# B&R Automation Studio project FeederLib (part 2)

#### FBFeeder.st
```iecst
(* TODO: Add your comment here *)
FUNCTION_BLOCK FBFeeder
	IF Enable THEN
		CASE Status OF
			FEED_ERROR:
			FEED_INIT:
				FBControl.Enable := TRUE;
				FBControl.TareK := Config.DefaultTareK;

				TON_BufferDelay.PT := Config.BufferDelay;
				TON_TareCalcDelay.PT := Config.TareCalcDelay;
				TON_DeviationCalcDelay.PT := Config.DeviationCalcDelay;
				TON_ToGoToAutoDelay.PT := Config.ToGoToAutoDelay;

				i := 0;
				j := 0;

				UserInfo.Rate := 0;
				UserInfo.TareK := 0;
				UserInfo.Deviation := 0;
				IF FBControl.Status = FEEDCTRL_READY_TO_FEED THEN
					Status := FEED_READY;
				END_IF
			FEED_READY:
				IF Start THEN
					FBControl.Start := TRUE;
				END_IF
				IF Reset THEN
					Status := FEED_RESET;
				END_IF
				IF FBControl.Status = FEEDCTRL_FEEDING THEN
					Status := FEED_FEEDING;
				END_IF
			FEED_FEEDING:
				IF Start THEN
					TON_WriteInBufferPeriod.IN := TRUE;
					TON_WriteInBufferPeriod();
					IF TON_WriteInBufferPeriod.Q THEN
						TON_WriteInBufferPeriod.IN := FALSE;
						IF NOT WriteInWTP THEN
							// задержка заполнения буфферов W T P
							TON_BufferDelay.IN := TRUE;
							TON_BufferDelay();
							IF TON_BufferDelay.Q THEN
								WriteInWTP := TRUE;
								TON_BufferDelay.IN := FALSE;
							END_IF
						ELSE
							// заполнение буфера W T P
							WBuffer[i] := UserInfo.Weight;
							IF i = 0 THEN
								PBuffer[0] := PBuffer[2399] + FBControl.UserInfo.ActualSpeed/100000;
								TBuffer[0] := TBuffer[2399] + 0.1;
							ELSE
								PBuffer[i] := PBuffer[i-1] + FBControl.UserInfo.ActualSpeed/100000;
								TBuffer[i] := TBuffer[i-1] + 0.1;
							END_IF

							IF i = 2399 THEN
								i := 0;
								RewriteWTP := TRUE;
							ELSE
								i := i + 1;
							END_IF

							IF NOT WriteInTareK THEN
								// задержка заполнения буффера тарировочного коэффициента
								TON_TareCalcDelay.IN := TRUE;
								TON_TareCalcDelay();
								IF TON_TareCalcDelay.Q THEN
									WriteInTareK := TRUE;
									TON_TareCalcDelay.IN := FALSE;
								END_IF
							ELSE
								// заполнение буффера тарировочного коэффициента
								IF RewriteWTP THEN
									UserInfo.TareK := USINT_TO_REAL(Config.Handler.Ratio)*FFeederRatio(ADR(WBuffer),ADR(PBuffer),ADR(TBuffer),2399)/0.6;
								ELSE
									UserInfo.TareK := USINT_TO_REAL(Config.Handler.Ratio)*FFeederRatio(ADR(WBuffer),ADR(PBuffer),ADR(TBuffer),i)/0.6;
								END_IF
								TareKBuffer[j] := UserInfo.TareK;

								IF j = 2399 THEN
									j := 0;
									RewriteTareK := TRUE;
								ELSE
									j := j + 1;
								END_IF

								IF NOT CalcDeviation THEN
									// задержка расчета стандартной погрешности татировочного коэффициента
									TON_DeviationCalcDelay.IN := TRUE;
									TON_DeviationCalcDelay();
									IF TON_DeviationCalcDelay.Q THEN
										CalcDeviation := TRUE;
										TON_DeviationCalcDelay.IN := FALSE;
									END_IF
								ELSE
									// расчет стандартного откланения погрешности тарировочного коэффициента
									IF RewriteTareK THEN
										UserInfo.Deviation := FStdDeviation(ADR(TareKBuffer),2399);
									ELSE
										UserInfo.Deviation := FStdDeviation(ADR(TareKBuffer),j);
									END_IF
								END_IF
							END_IF
						END_IF
					END_IF
					// Выбор тарировочного коэффициента в зависимости от конфигурации
					IF Control.ManualTareControl THEN
						FBControl.TareK := Control.TareK;
					ELSE
						IF NOT UserInfo.IsAUTO THEN
							FBControl.TareK := Config.DefaultTareK;
							IF CalcDeviation THEN
								IF (UserInfo.Deviation <> 0) AND (UserInfo.Deviation < Config.DeviationLimit) THEN
									TON_ToGoToAutoDelay.IN := TRUE;
									IF TON_ToGoToAutoDelay.Q THEN
										UserInfo.IsAUTO := TRUE;
										TON_ToGoToAutoDelay.IN := FALSE;
									END_IF;
								ELSE
									TON_ToGoToAutoDelay.IN := FALSE;
									FBControl.TareK := Config.DefaultTareK;
								END_IF
								TON_ToGoToAutoDelay();
							ELSE
								FBControl.TareK := Config.DefaultTareK;
							END_IF
						ELSE
							IF UserInfo.Deviation < Config.DeviationLimit THEN
								UserInfo.IsAUTO := FALSE;
							ELSE
								FBControl.TareK := UserInfo.TareK;
							END_IF
						END_IF
					END_IF
				ELSE
					FBControl.Start := FALSE;
					Status := FEED_PAUSE;
				END_IF
			FEED_RESET:
				FOR i := 0 TO 2399 DO
					WBuffer[i] := 0;
					TBuffer[i] := 0;
					PBuffer[i] := 0;
					TareKBuffer[i] := 0;
				END_FOR
				i := 0;
				j := 0;

				RewriteWTP := FALSE;
				RewriteTareK := FALSE;
				WriteInWTP := FALSE;
				WriteInTareK := FALSE;
				CalcDeviation := FALSE;
				UserInfo.IsAUTO := FALSE;

				Reset := FALSE;
				Status := FEED_READY;

				UserInfo.Rate := 0;
				UserInfo.TareK := 0;
				UserInfo.Deviation := 0;
			FEED_PAUSE:
				IF Start THEN
					Status := FEED_READY;
					IF RewriteWTP THEN
						IF i = 0 THEN
							IF ABS(WBuffer[2399]-UserInfo.Weight) > Config.ResetWeightLimit THEN
								Status := FEED_RESET;
							END_IF
						ELSE
							IF ABS(WBuffer[i-1]-UserInfo.Weight) > Config.ResetWeightLimit THEN
								Status := FEED_RESET;
							END_IF
						END_IF
					ELSE
						IF (i <> 0) AND (ABS(WBuffer[i-1]-UserInfo.Weight) > Config.ResetWeightLimit) THEN
							Status := FEED_RESET;
						END_IF
					END_IF
				END_IF
		END_CASE
		FBControl.Config := Config.Handler;
		FBControl.Control := Control.Handler;
		FBControl.IOin := IOin.Handler;
		FBControl();
		UserInfo.Handler := FBControl.UserInfo;
		UserInfo.Weight := CalibrateREAL(DINT_TO_REAL(IOin.aiWeight), Config.WeightCalibrate);
		UserInfo.Rate := FBControl.UserInfo.ActualSpeed*UserInfo.TareK*0.6/USINT_TO_REAL(Config.Handler.Ratio);
		IOout := FBControl.IOout;
	ELSE
		Status := FEED_INIT;
	END_IF
END_FUNCTION_BLOCK
```

#### FBFeederHandler.st
```iecst
(* TODO: Add your comment here *)
FUNCTION_BLOCK FBFeederHandler
	IF Enable THEN
		CASE Status OF
			FEEDCTRL_ERROR:
				// error case
			FEEDCTRL_INIT:
				AxisBasic.MpLink := Config.AxisConfigLink;
				AxisBasic.Enable := TRUE;
				AxisBasic.Parameters := Config.AxisBasicParLink;
				AxisBasic.Axis := Config.ACPConfigLink;

				AxisCyclicSet.MpLink := Config.AxisConfigLink;
				AxisCyclicSet.Enable := TRUE;
				AxisCyclicSet.Parameters := Config.AxisCyclicSetParLink;

				IF (AxisBasic.Active) THEN
					UserInfo.Active := TRUE;
					AxisBasic.Power := 1;
					IF (AxisBasic.PowerOn) THEN
						IF (AxisBasic.IsHomed = 0) THEN
							AxisBasic.Home := 1;
						ELSE
							AxisBasic.Home := 0;
							IF (AxisCyclicSet.Active) THEN
								AxisCyclicSet.CyclicVelocity := 1;
								Status := FEEDCTRL_READY_TO_FEED;
							END_IF
						END_IF
					END_IF
				END_IF

			FEEDCTRL_READY_TO_FEED:
				IF (Start) THEN
					Status := FEEDCTRL_PREPURGE;
				END_IF

				IOout.aoGasRate := 0;
				IOout.doShutOff := TRUE;
				IOout.doMixer := FALSE;
			FEEDCTRL_PREPURGE:
				IF (Start) THEN
					IF (TON_Prepurge.Q) THEN
						TON_Prepurge.IN := 0;
						Status := FEEDCTRL_FEEDING;
					ELSE
						TON_Prepurge.IN := 1;
					END_IF
				ELSE
					TON_Prepurge.IN := 0;
					Status := FEEDCTRL_READY_TO_FEED;
				END_IF
				TON_Prepurge(PT := Config.PrepurgeTime);

				IOout.aoGasRate := Calibrate(Control.GasRate,Config.GasCalibrateOut);
				IOout.doShutOff := FALSE;
				IOout.doMixer := TRUE;
			FEEDCTRL_FEEDING:
				IF (Start) THEN
					AxisCyclicSet.Velocity := ((LIMIT(0,(Control.PowderRate/(TareK*10)),100)*(100+Control.KZU))/Control.KZP)*Config.Ratio/0.6;
				ELSE
					AxisCyclicSet.Velocity := 0;
					Status := FEEDCTRL_POSTPURGE;
				END_IF

				IOout.aoGasRate := Calibrate(Control.GasRate,Config.GasCalibrateOut);
			FEEDCTRL_POSTPURGE:
				IF (Start) THEN
					TON_Postpurge.IN := 0;
					Status := FEEDCTRL_FEEDING;
				ELSE
					IF (TON_Postpurge.Q) THEN
						TON_Postpurge.IN := 0;
						Status := FEEDCTRL_READY_TO_FEED;
					ELSE
						TON_Postpurge.IN := 1;
					END_IF
				END_IF
				TON_Postpurge(PT := Config.PostpurgeTime);

				IOout.aoGasRate := Calibrate(Control.GasRate,Config.GasCalibrateOut);
		END_CASE
		// добавить проверку чтобы AxisConfigLink != 0
		AxisBasic();
		AxisCyclicSet();

		UserInfo.ActualSpeed := AxisBasic.Velocity;
	END_IF

END_FUNCTION_BLOCK
```

#### FBSpendTotalizer.st
```iecst
(* TODO: Add your comment here *)
FUNCTION_BLOCK FBSpendTotalizer

	CASE Status OF
		SPENDTOTALIZER_INIT:
			TON_WeightCheckPeriod.PT := Period;
			Status := SPENDTOTALIZER_WAIT;
		SPENDTOTALIZER_BIZY:
			TON_WeightCheckPeriod();
			IF TON_WeightCheckPeriod.Q THEN
				IF ((TempVal - Weight) > Delta) AND ((TempVal - Weight) > 0) THEN
					CounterLink := CounterLink + (TempVal - Weight);
					TempVal := Weight;
				END_IF
				TON_WeightCheckPeriod.IN := FALSE;
				TON_WeightCheckPeriod();
				TON_WeightCheckPeriod.IN := TRUE;
			END_IF
			IF NOT Active THEN
				IF ((TempVal - Weight) < Delta) AND ((TempVal - Weight) > 0) THEN
					CounterLink := CounterLink + (TempVal - Weight);
					TempVal := Weight;
				END_IF
				TON_WeightCheckPeriod.IN := FALSE;
				TON_WeightCheckPeriod();
				Status := SPENDTOTALIZER_PAUSE;
			END_IF
		SPENDTOTALIZER_PAUSE:
			IF Active THEN
				IF (ABS(TempVal - Weight) > 10*Delta) THEN
					Status := SPENDTOTALIZER_WAIT;
				ELSE
					Status := SPENDTOTALIZER_BIZY;
				END_IF
			END_IF
			TON_WeightCheckPeriod.IN := TRUE;
		SPENDTOTALIZER_WAIT:
			IF Active THEN
				TempVal := Weight;
				Status := SPENDTOTALIZER_BIZY;
			END_IF
	END_CASE

END_FUNCTION_BLOCK
```

#### FBFeederControl.st - not listed in the package file held
```iecst
(* TODO: Add your comment here *)
FUNCTION_BLOCK FBFeederControl
	IF Enable THEN
		CASE Status OF
			FEEDCTRL_ERROR:
				// error case
			FEEDCTRL_INIT:
				// добавить проверку чтобы AxisConfigLink != 0
				AxisBasic.MpLink := Config.AxisConfigLink;
				AxisBasic.Enable := TRUE;
				AxisBasic.Parameters := Config.AxisBasicParLink;
				AxisBasic.Axis := Config.ACPConfigLink;

				AxisCyclicSet.MpLink := Config.AxisConfigLink;
				AxisCyclicSet.Enable := TRUE;
				AxisCyclicSet.Parameters := Config.AxisCyclicSetParLink;

				IF (AxisBasic.Active) THEN
					UserInfo.Active := TRUE;
					AxisBasic.Power := 1;
					IF (AxisBasic.PowerOn) THEN
						IF (AxisBasic.IsHomed = 0) THEN
							AxisBasic.Home := 1;
						ELSE
							AxisBasic.Home := 0;
							IF (AxisCyclicSet.Active) THEN
								AxisCyclicSet.CyclicVelocity := 1;
								Status := FEEDCTRL_READY_TO_FEED;
							END_IF;
						END_IF;
					END_IF;
				END_IF;
			FEEDCTRL_READY_TO_FEED:
				IF (Start) THEN
					Status := FEEDCTRL_PREPURGE;
				END_IF

				IO.Out.aoGasRate := 0;
				IO.Out.doShutOff := TRUE;
				IO.Out.doMixer := FALSE;
			FEEDCTRL_PREPURGE:
				IF (Start) THEN
					IF (TON_Prepurge.Q) THEN
						TON_Prepurge.IN := 0;
						Status := FEEDCTRL_FEEDING;
					ELSE
						TON_Prepurge.IN := 1;
					END_IF
				ELSE
					TON_Prepurge.IN := 0;
					Status := FEEDCTRL_READY_TO_FEED;
				END_IF
				TON_Prepurge(PT := Config.PrepurgeTime);

				IO.Out.aoGasRate := Calibrate(Control.GasRate,Config.GasCalibrateOut);
				IO.Out.doShutOff := FALSE;
				IO.Out.doMixer := TRUE;
			FEEDCTRL_FEEDING:
				IF (Start) THEN
					AxisCyclicSet.Velocity := ((Control.PowderRate*(100+Control.KZU))/Control.KZP)*TareK;
				ELSE
					AxisCyclicSet.Velocity := 0;
					Status := FEEDCTRL_POSTPURGE;
				END_IF

				IO.Out.aoGasRate := Calibrate(Control.GasRate,Config.GasCalibrateOut);
			FEEDCTRL_POSTPURGE:
				IF (Start) THEN
					TON_Postpurge.IN := 0;
					Status := FEEDCTRL_FEEDING;
				ELSE
					IF (TON_Postpurge.Q) THEN
						TON_Postpurge.IN := 0;
						Status := FEEDCTRL_READY_TO_FEED;
					ELSE
						TON_Postpurge.IN := 1;
					END_IF
				END_IF
				TON_Postpurge(PT := Config.PostpurgeTime);

				IO.Out.aoGasRate := Calibrate(Control.GasRate,Config.GasCalibrateOut);
		END_CASE
		AxisBasic();
		AxisCyclicSet();
		UserInfo.ActualSpeed := AxisBasic.Velocity;
	END_IF

END_FUNCTION_BLOCK
```

#### FLinearRegrationKoef.st - not listed in the package file held
```iecst
(* TODO: Add your comment here *)
FUNCTION FLinearRegrationKoef
	sumx := 0;
	sumy := 0;
	sump := 0;
	sumx2 := 0;
	sumxy := 0;
	sumxp := 0;

	FOR i := 0 TO n-1 DO
		weight ACCESS (weightArrayAdr + 32*i);
		position ACCESS (positionArrayAdr + 32*i);
		sumy := sumy + weight;
		sump := sump + position;
		sumxy := sumxy + (i*weight);
		sumxp := sumxp + (i*position);
	END_FOR
	sumx := (lengthOfArray*(lengthOfArray+1))/2;
	sumx2 := (lengthOfArray*(lengthOfArray+1)*(2*lengthOfArray+1))/6;

	sxx := sumx2 - (sumx*sumx)/UINT_TO_REAL(n);
	sxy := sumxy - (sumx*sumy)/UINT_TO_REAL(n);
	sxp := sumxp - (sumx*sump)/UINT_TO_REAL(n);
	k := sxy/sxx;
	kp := sxp/sxx;

	FLinearRegrationKoef := (-k*60)/kp;
END_FUNCTION
```

#### FRatePerMinute.st - not listed in the package file held
```iecst
(* TODO: Add your comment here *)
FUNCTION FRatePerMinute
	sumx := 0;
	sumy := 0;
	sump := 0;
	sumx2 := 0;
	sumxy := 0;
	sumxp := 0;

	FOR i := 0 TO lengthOfArray-1 DO
		sumy := sumy + W[i];
		sump := sump + V[i];
		sumxy := sumxy + (i*W[i])*(UDINT_TO_LREAL(i+1)/1000);
		sumxp := sumxp + (i*W[i])*(UDINT_TO_LREAL(i+1)/1000);
	END_FOR
	sumx := ((lengthOfArray*(lengthOfArray+1))/2)/1000;
	sumx2 := (((lengthOfArray/10000)*((lengthOfArray+1)/10000)*((2*lengthOfArray+1)/10000))/6);

	sxx := sumx2 - (sumx*sumx)/UDINT_TO_REAL(lengthOfArray);
	sxy := sumxy - (sumx*sumy)/UDINT_TO_REAL(lengthOfArray);
	sxp := sumxp - (sumx*sump)/UDINT_TO_REAL(lengthOfArray);
//	k := sxy/sxx;
//	kp := sxp/sxx;

	FRatePerMinute := LREAL_TO_REAL(((sxy/sxx)*10)/(sxp/sxx));
END_FUNCTION
```

### Program Logical/Program (IEC)

#### Main.st - Init, cyclic, exit code
```iecst
PROGRAM _INIT
	tempStr := '';
	RD.DeviceName := 'HardDisk';
	RD.FileName := 'TestFile1';
	RD.Ena := FALSE;
	RD.Offset := 0;
	RD.Size := 1;
	i := 0;
END_PROGRAM

PROGRAM _CYCLIC

	IF Start THEN
		RD();
		tempStr := RD.Symbol;
		Start := FALSE;
	END_IF

END_PROGRAM

PROGRAM _EXIT
(* Insert code here *)

END_PROGRAM
```

#### Variables.var - Local variables
```iecst
VAR
	RD : FB_ReadData;
	tempStr : STRING[80];
	Start : BOOL := FALSE;
	T : REAL;
	W : ARRAY[0..2399] OF REAL := [2400(0)];
	V : ARRAY[0..2399] OF REAL := [2400(0)];
	RT : REAL;
	KT : REAL;
	i : UDINT;
	override : BOOL;
	Ktare : REAL;
	Weight : REAL;
END_VAR
```

#### LocalFunctions.fun
```iecst
FUNCTION_BLOCK FB_ReadData
	VAR_INPUT RETAIN
		Ena : BOOL := FALSE;
		FileName : STRING[32];
		DeviceName : STRING[32];
	END_VAR
	VAR_INPUT
		Offset : UDINT := 0;
		Size : UDINT := 1;
	END_VAR
	VAR_OUTPUT
		Status : STRING[80]; (*0-ok*)
		Symbol : STRING[80];
		wStatus : UINT;
	END_VAR
	VAR
		FOpen : FileOpen;
		FRead : FileRead;
		FClose : FileClose;
		Enable_trig : R_TRIG; (*Триггер старта расчета расхода*)
		Disable_trig : F_TRIG; (*Триггер остановки расчета расхода*)
		dwIdent : UDINT;
	END_VAR
END_FUNCTION_BLOCK
```

#### ReadData.st
```iecst
(* TODO: Add your comment here *)
FUNCTION_BLOCK FB_ReadData
	Enable_trig(CLK := Ena);
	Disable_trig(CLK := Ena);

	IF Enable_trig.Q THEN
		IF (FileName = '') OR (DeviceName = '') THEN
			Ena := FALSE;
			Status := 'Incorrect FileName or DeviceName';
		ELSE
			Status := '';

			(**** Try to open existing file ****)
			FOpen.enable    := 1;
			FOpen.pDevice   := ADR(DeviceName);
			FOpen.pFile     := ADR(FileName);
			FOpen.mode      := FILE_RW;  (* Read and write access *)
			(* Call FBK *)
			FOpen();
			(* Get FBK output information *)
			dwIdent := FOpen.ident;
			wStatus := FOpen.status;
			(* Verify status (20708 -> File doesn't exist) *)
			IF (wStatus = 20708) THEN
				Status := 'File doesnt exist';
			ELSE
				IF (wStatus = 0) THEN
					Status := 'OK';
				ELSE
					IF (wStatus <> 65535) THEN

						Status := 'Open file error';

					END_IF
				END_IF
			END_IF
		END_IF
	ELSE
		IF Ena THEN
			IF ((Offset + Size) > FOpen.filelen) THEN
				Status := 'EOF';
				wStatus := 5;
				Ena := FALSE;
			ELSE
				(**** Read data from file ****)
				(* Initialize file read structure *)
				FRead.enable    := 1;
				FRead.ident     := dwIdent;
				FRead.offset    := Offset;
				FRead.pDest     := ADR(Symbol);
				FRead.len       := Size;
				(* Call FBK *)
				FRead();
				(* Get status *)
				wStatus := FRead.status;
				(* Verify status *)
				IF (wStatus = 0) THEN
					Status := 'OK';
					Offset := Offset + Size;
				ELSE
					IF (wStatus <> 65535) THEN
						Status := 'Reading file error';
						Ena := FALSE;
					END_IF
				END_IF
			END_IF
		END_IF
	END_IF

	IF Disable_trig.Q OR (wStatus = 5) THEN
		(**** Close file ****)
		(* Initialize file close structure *)
		FClose.enable   := 1;
		FClose.ident    := dwIdent;
		(* Call FBK *)
		FClose();
		(* Get status *)
		wStatus := FClose.status;
		Offset := 0;
		(* Verify status *)
		//			IF (wStatus = 0) THEN
		//				byStep := 6;
		//			ELSE
		//				IF (wStatus <> 65535) THEN
		//					byErrorLevel := 5;
		//					byStep := 0;
		//					IF (wStatus = 20799) THEN
		//						wError := FileIoGetSysError();
		//					END_IF
		//				END_IF
		//			END_IF
	END_IF

END_FUNCTION_BLOCK
```

### Program Logical/ReadTest

#### Variables.var
```iecst
VAR
	FBRead1 : FBReadFromFile;
	ReadedStr : STRING[80];
	ReadedValue : REAL;
	Offset : UDINT;
	Read : BOOL;
	TempString : STRING[80];
	i : UDINT;
END_VAR
```

#### Main.st
```iecst
PROGRAM _INIT
	(* Insert code here *)
	FBRead1.Enable := TRUE;
	FBRead1.strDevice := 'HardDisk';
	FBRead1.strFile := 'TestFile1';
	FBRead1.BytesToRead := 1;
	Offset := 0;
	FBRead1.Offset := Offset;
	TempString := '';
	i := 0;
END_PROGRAM

PROGRAM _CYCLIC
	(* Insert code here *)
//	WHILE Read DO
			IF Read THEN
		FBRead1.Read := TRUE;
		FBRead1.Offset := Offset;
		i:= i+1;
		FBRead1();
		IF (FBRead1.byStep = 3) THEN
			IF (FBRead1.ReadedStr <> ',') THEN
				IF (FBRead1.wStatus <> 65535) THEN
					IF (FBRead1.wStatus = 0) THEN
						IF (FBRead1.ReadedStr <> '$n') OR (FBRead1.ReadedStr <> '$r') THEN
							TempString := CONCAT(TempString,FBRead1.ReadedStr);
						END_IF
						Offset := Offset + 1;
						FBRead1();
					ELSE
						//					Read := FALSE;
						//					FBRead1.Enable := FALSE;
						//					TempString := '';
						FBRead1();
					END_IF
				ELSE
					FBRead1();
				END_IF
			ELSE
				Read := FALSE;
				FBRead1.Read := FALSE;
				Offset := Offset + 1;
				ReadedValue := STRING_TO_REAL(TempString);
				TempString := '';
			END_IF
		END_IF
//	END_WHILE
		END_IF
END_PROGRAM

PROGRAM _EXIT
			(* Insert code here *)

END_PROGRAM
```

Listed in the project but not available here: Logical/Global.typ, Logical/Libraries/UserLib/Constants.var, Logical/ReadData/Types.typ, Logical/gAxis02obj, Logical/FeederLib/Constants.var, Logical/Program/Types.typ
